# B&R Automation Studio project DietrichBrewing
Automation Studio 4.12.3.127 SP; technology packages: Acp10Arnc0 5.19.1, mapp 5.19.0, mappControl 5.19.0, mappView 5.19.0

## Configuration Config1

CPU X20CP0482, AutomationRuntime B4.93, Build 4.1.2, Safety 0.0, Vc V4.72.6

### Task classes (Cpu.sw)
```
Cyclic#1 (cycle 1000 us, tolerance 0 us):
  KettleCont <- ProcessControl.KettleControl.prg
Cyclic#2 (cycle 20000 us, tolerance 20000 us):
  HLTControl <- ProcessControl.HLTControl.prg
Cyclic#4 (cycle 100000 us, tolerance 100000 us):
  BrewingSeq <- Brewing.BrewingSeq.prg
  HMIProgram <- HMIControl.HMIProgram.prg
  MashTunCon <- ProcessControl.MashTunControl.prg
Binaries: FWRules, arsvcreg, TCData, udbdef, mvLoader, User, iomap, Config, Role, arconfig, asfw, ashwac, sysconf, ashwd, Config_1
Libraries: MpTemp, MpBase, MTBasics, brsystem, sys_lib, MTTypes, runtime, Functions, standard, asieccon, arssl, AsIODiag, Acp10man, Acp10par, NcGlobal, ViBase, AsZip, FileIO, AsARCfg, powerlnk, AsEPL, AsIO, astime, SfDomain, CoTrace
```

### Hardware
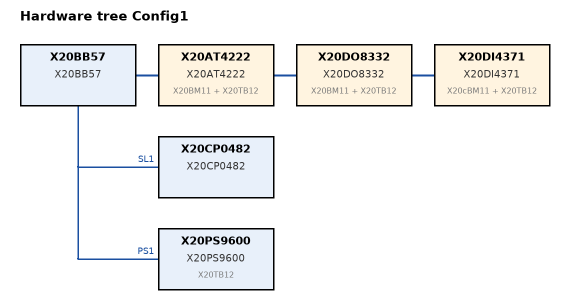
```
X20AT4222 : X20AT4222 v1.4.0.0  [SS1 -> X20TB12a.SS; SL -> X20BM11.SL1]
  InputFilter = 1ms
X20BB57 : X20BB57 v1.2.0.0
X20BM11 : X20BM11 v1.1.0.0  [X2X1 -> X20BB57.IF6]
X20BM11a : X20BM11 v1.1.0.0  [X2X1 -> X20BM11.X2X2]
X20CP0482 : X20CP0482 v1.7.0.0  [SL -> X20BB57.SL1]
  Connector IF2:
    ActivateDevice = 1
    Mode = Manual
    InternetAddress = 192.168.4.64
    SubnetMask = 255.255.255.0
  Connector IF3:
    ActivatePowerlink = 0
  ConfigurationID = DietrichBrewing_Config1
  TimerDeviceType = SWIOTIMER
  SystemTick = 1000
  Cyclic1Duration = 1000
  Cyclic1Tolerance = 0
  Cyclic2Duration = 20000
  Cyclic2Tolerance = 20000
  Cyclic3Duration = 50000
  Cyclic3Tolerance = 50000
  Cyclic4Duration = 100000
  Cyclic4Tolerance = 100000
  Cyclic5Duration = 200000
  Cyclic5Tolerance = 200000
  Cyclic6Duration = 500000
  Cyclic6Tolerance = 500000
  Cyclic7Duration = 1000000
  Cyclic7Tolerance = 1000000
  Cyclic8Duration = 10000
  Cyclic8Tolerance = 30000000
  FileDevice1
  FileDeviceName1 = USER
  FileDevicePath1 = USER_PATH
  ActivateOpcUa = 1
  OpcUaInformationModels_PV_Version = 1
X20DI4371 : X20DI4371 v1.2.0.0  [SS1 -> X20TB12c.SS; SL -> X20cBM11.SL1]
  Supervision = off
X20DO8332 : X20DO8332 v1.5.0.0  [SS1 -> X20TB12b.SS; SL -> X20BM11a.SL1]
X20PS9600 : X20PS9600 v1.6.0.0  [PS -> X20BB57.PS1; SS1 -> X20TB12.SS]
X20TB12 : X20TB12 v1.0.0.0
X20TB12a : X20TB12 v1.0.0.0
X20TB12b : X20TB12 v1.0.0.0
X20TB12c : X20TB12 v1.0.0.0
X20cBM11 : X20cBM11 v1.1.0.0  [X2X1 -> X20BM11a.X2X2]
```

### IoMap.iom - X20CP0482/IoMap.iom
```iecst
VAR_CONFIG
	::HLTHeater AT %QX."X20DO8332".DigitalOutput01;
	::KettleHeater AT %QX."X20DO8332".DigitalOutput02;
	::HLTPump AT %QX."X20DO8332".DigitalOutput03;
	::MashPump AT %QX."X20DO8332".DigitalOutput04;
	::Buzzer AT %QX."X20DO8332".DigitalOutput05;
	::ValveSelector AT %QX."X20DO8332".DigitalOutput06;
	::ValveOff AT %QX."X20DO8332".DigitalOutput07;
	::ValveOn AT %QX."X20DO8332".DigitalOutput08;
END_VAR
```

### Acp10cfg.ncc - X20CP0482/Motion/Acp10cfg.ncc
```
NcConfiguration (Version=5.16.2, NcSwId=Acp10)
  ACP10CF1_typ:
    cnt_nettrc_rec_drive = 150
    bufsize_trace_upload = 1200
    tc_nc_man_task = Cyclic #1
    glob_pv_as_ncobject = Yes
    ncsys_dl_broadcast = Yes
    ncsys_dl_acp_reset = Yes
    safemc_log_err_to_ax = Yes
    network_init:
      ncsw_init_execute = Yes
      automatic_execute = No
      node_nr_warning = Yes
      net_err_before_ncact = Yes
    nettrc:
      enter_parsecrec = Yes
      enter_ncaction = Yes
      save_ring_startidx = No
    cam_prof_download:
      cam_dat_dl_parallel = No
      tc_cam_dl_parallel = Task class for NC Manager task
```

### Config.tempcontroller - X20CP0482/mappControl/Config.tempcontroller
```
Element Cfg_HLTTemp (Type=tempcontroller)
  TempController:
    PWMParameters:
      Heat:
        Period = 0.5
  Alarms:
    UserAlarm = Yes
Element Cfg_KettleTemp (Type=tempcontroller)
  Alarms:
    UserAlarm = Yes
```

## Logical view

Binary libraries used (declarations not repeated): operator, runtime, astime, AsIecCon, brsystem, sys_lib, MTTypes, standard, AsIODiag, ViBase, AsZip, FileIO, AsARCfg, powerlnk, AsEPL, AsIO, CoTrace, Acp10man 5.19.1, Acp10par 5.19.1, NcGlobal 5.19.1, MpAlarmX, MpBase, MpTemp 5.19.0, MTBasics

### Global.typ - Global data types
```iecst
(*Main Type*)

TYPE
	MashToHLT : 	STRUCT
		Start : BOOL;
		HLTTemp : REAL;
	END_STRUCT;
	ProcControl : 	STRUCT
		setPower : REAL;
		currPower : REAL;
		currTemp : REAL;
		SetTemp : REAL;
		TempCtrl : TempCont;
		State : ControlState;
		Status : SystemStatus;
		i : SystemInput;
	END_STRUCT;
END_TYPE

(*HMI Inputs and Status*)

TYPE
	SystemInput : 	STRUCT
		ResetError : BOOL;
		EStop : BOOL;
		Auto : BOOL;
		Stop : BOOL;
		Pause : BOOL;
		Start : BOOL;
	END_STRUCT;
	SystemStatus : 	STRUCT
		Automatic : BOOL;
		Manual : BOOL;
		Running : BOOL;
		Stopped : BOOL;
		Paused : BOOL;
		On : BOOL;
	END_STRUCT;
END_TYPE

(*Temp Controller Types*)

TYPE
	TempCont : 	STRUCT
		Ctrl : MpTempController;
		Ptr : MpTempControllerParType;
		PWM : MTBasicsPWM;
	END_STRUCT;
END_TYPE

(*State Machines*)

TYPE
	ControlState :
		(
		Stop,
		Manual,
		Automatic
		);
END_TYPE
```

### Global.var - Global variables
```iecst
(*Between Programs*)
VAR
	FromMashCyc : MashToHLT;
END_VAR
(*Output Mapping*)
VAR
	Buzzer : BOOL;
	ValveSelector : BOOL; (*Off = Mash, On = HLT*)
	ValveOff : BOOL;
	ValveOn : BOOL;
	SysPower : BOOL;
	HLTPump : BOOL;
	MashPump : BOOL;
	CoolingPump : BOOL;
	HLTHeater : BOOL;
	KettleHeater : BOOL;
END_VAR
(*Temperature Controller Variables*)
VAR
	rawMashTemp : INT;
	rawKettleTemp : INT;
	rawHLTTemp : INT;
END_VAR
```

### Package Logical/Libraries - Global libraries

### Library Logical/Libraries/Functions (IEC)

#### Functions.fun - Exported functions and function blocks
```iecst
{REDUND_ERROR} FUNCTION Device : BOOL (*TODO: Add your comment here*) (*$GROUP=User,$CAT=User,$GROUPICON=User.png,$CATICON=User.png*)
	VAR_INPUT
		AutoMode : BOOL;
		AutoExpected : BOOL;
		pbExpected : BOOL;
	END_VAR
	VAR_IN_OUT
		Output : BOOL;
	END_VAR
	VAR
		Expected : BOOL;
	END_VAR
END_FUNCTION
```

#### Device.st
```iecst
//Set device on or off with HMI or sequence
FUNCTION Device

	IF NOT AutoMode THEN

		//Manual Operation
		IF pbExpected  THEN
			Expected  := TRUE;
		ELSIF NOT pbExpected THEN
			Expected  := FALSE;
		END_IF

	ELSE
		//Auto operation
		IF AutoExpected THEN
			Expected:= TRUE;
		ELSIF NOT AutoExpected THEN
			Expected := FALSE;
		END_IF
	END_IF

	//Set output of function
	Output := Expected;
END_FUNCTION
```

### Program Logical/Brewing/BrewingSeq (IEC)

#### Types.typ
```iecst
TYPE
	Seq :
		(
		Reset,
		FillTanks,
		PreHeat,
		Mash,
		Boil
		);
END_TYPE
```

#### Variables.var
```iecst
VAR
	HeatTime : TON;
	Sequence : Seq;
	pbMashPump : BOOL;
END_VAR
```

#### Main.st
```iecst
PROGRAM _INIT

END_PROGRAM

PROGRAM _CYCLIC

END_PROGRAM

PROGRAM _EXIT
	(* Insert code here *)

END_PROGRAM
```

### Program Logical/Brewing/HLTControl

#### Variables.var
```iecst
VAR
	PumpExp : BOOL;
	Proc : ProcControl;
END_VAR
```

#### Main.st
```iecst
PROGRAM _INIT

END_PROGRAM

PROGRAM _CYCLIC
	//Initilize Temp Controller FB
	Proc.TempCtrl.Ctrl.Parameters := ADR(Proc.TempCtrl.Ptr);
	Proc.TempCtrl.Ctrl.MpLink := ADR(Cfg_HLTTemp);

	//Mash cycle variables
	IF EDGEPOS(FromMashCyc.Start) THEN
		Proc.i.Auto 	:= TRUE;
		Proc.i.Start 	:= TRUE;
		Proc.SetTemp 	:= FromMashCyc.HLTTemp;
	ELSIF EDGENEG(FromMashCyc.Start) THEN
		Proc.i.Auto 	:= FALSE;
		Proc.i.Start 	:= FALSE;
	END_IF

	//Automatic and manual conditions
	Proc.Status.Automatic 	:= Proc.i.Auto;
	Proc.Status.Manual		:= NOT Proc.i.Auto;

	//Map Variables
	Proc.TempCtrl.Ctrl.Control := Proc.i.Start;
	Proc.TempCtrl.Ctrl.ErrorReset := Proc.i.ResetError;
	Proc.TempCtrl.Ctrl.SetTemperature := Proc.SetTemp;

	IF Proc.Status.Automatic THEN
		Proc.State := Automatic;
	ELSIF Proc.Status.Manual THEN
		Proc.State := Manual;
	END_IF

	//Set the state machine
	IF  DiagCpuIsARsim() OR DiagCpuIsSimulated() THEN
		Proc.currTemp := Proc.TempCtrl.Ctrl.Info.Simulation.ActualTemperature;
		Proc.currPower := Proc.TempCtrl.Ctrl.Info.Simulation.HeatValue;
		Proc.TempCtrl.Ctrl.Simulate := TRUE;
	ELSE
		Proc.TempCtrl.Ctrl.ActualTemperature := rawHLTTemp * 1000;

		Proc.currTemp	:= rawHLTTemp * 1000;
		Proc.TempCtrl.Ctrl.Simulate := FALSE;
	END_IF

	//Temperature controller state machine
	CASE Proc.State OF

		Automatic:
			//Temperature control parameters
			Proc.TempCtrl.PWM.Enable 	:= FALSE;
			Proc.TempCtrl.Ctrl.Enable 	:= TRUE;

			//HMI Variables
			HLTHeater := Proc.TempCtrl.Ctrl.Heat;
			Proc.currPower 	:= Proc.TempCtrl.Ctrl.HeatValue;

		Manual:
			//Temperature control parmeters
			Proc.TempCtrl.PWM.Enable 	:= Proc.i.Start;
			Proc.TempCtrl.Ctrl.Enable 	:= FALSE;
			Proc.TempCtrl.PWM.DutyCycle := Proc.setPower;
			Proc.TempCtrl.PWM.MinPulseWidth := 0.1;
			Proc.TempCtrl.PWM.Period := 1.0;

			//HMI Variables
			HLTHeater := Proc.TempCtrl.PWM.Out;
			IF Proc.TempCtrl.PWM.Active THEN
				Proc.currPower := Proc.TempCtrl.PWM.DutyCycle;
			ELSE
				Proc.currPower := 0;
			END_IF

	END_CASE

	//Call FB's
	Proc.TempCtrl.Ctrl();
	Proc.TempCtrl.PWM();

	//Set pump output
	HLTPump := PumpExp;
END_PROGRAM

PROGRAM _EXIT
	(* Insert code here *)

END_PROGRAM
```

### Program Logical/Brewing/KettleControl (IEC)

#### Main.st - Init, cyclic, exit code
```iecst
PROGRAM _INIT
	(* Insert code here *)

END_PROGRAM

PROGRAM _CYCLIC
	//Initilize Temp Controller FB
	Proc.TempCtrl.Ctrl.Parameters := ADR(Proc.TempCtrl.Ptr);
	Proc.TempCtrl.Ctrl.MpLink := ADR(Cfg_KettleTemp);
	//Map Variables
	Proc.TempCtrl.Ctrl.Control := Proc.i.Start;
	Proc.TempCtrl.Ctrl.ErrorReset := Proc.i.ResetError;

	//Automatic and manual conditions
	Proc.Status.Automatic 	:= Proc.i.Auto;
	Proc.Status.Manual		:= NOT Proc.i.Auto;

	IF Proc.Status.Automatic THEN
		Proc.State := Automatic;
	ELSIF Proc.Status.Manual THEN
		Proc.State := Manual;
	ELSE
	;
	END_IF

	//Set the state machine
	IF  DiagCpuIsARsim() OR DiagCpuIsSimulated() THEN
		Proc.TempCtrl.Ctrl.Enable	:= TRUE;
		Proc.TempCtrl.Ctrl.Simulate := TRUE;
		Proc.currTemp := Proc.TempCtrl.Ctrl.Info.Simulation.ActualTemperature;
	ELSE
		Proc.currTemp := rawHLTTemp * 1000;
	END_IF

	//Temperature controller state machine
	CASE Proc.State OF

		Manual:
			//PWM control
			Proc.TempCtrl.PWM.Enable 	:= Proc.i.Start;

			//PWM Parameters
			Proc.TempCtrl.PWM.DutyCycle := Proc.setPower;
			Proc.TempCtrl.PWM.MinPulseWidth := 0.1;
			Proc.TempCtrl.PWM.Period 		:= 1.0;
			KettleHeater := Proc.TempCtrl.PWM.Out;

			//HMI Variables
			IF Proc.TempCtrl.PWM.Active THEN
				Proc.currPower := Proc.TempCtrl.PWM.DutyCycle;
			ELSE
				Proc.currPower := 0;
			END_IF

		Automatic:
			//Not Used

	END_CASE

	//Call Action Files
	Displayclock;
	PowerControl;

	//Call FB's
	Proc.TempCtrl.Ctrl();
	Proc.TempCtrl.PWM();
	KettleTmr();
END_PROGRAM

PROGRAM _EXIT
	(* Insert code here *)

END_PROGRAM
```

#### Variables.var - Local variables
```iecst
(*Hop Control Variables*)
VAR
	SelectedHopTime : USINT;
	HopTime : ARRAY[0..5] OF USINT;
	i : INT;
	currHop : INT;
	remainTime : USINT;
END_VAR
(*Kettle Control*)
VAR
	Proc : ProcControl;
	KettleTmr : TON;
	TimePre : TIME;
	StartKettle : BOOL;
	TmrDT : TIMEStructure;
	HrRe : STRING[4];
	MinRe : STRING[4];
	SecRe : STRING[4];
	TmrRemain : STRING[10];
	pbFastDown : BOOL;
	pbFastUp : BOOL;
	pbUp : BOOL;
	pbDown : BOOL;
	HopSelection : DINT;
	PrevSelection : DINT;
	PrevHopTime : DINT;
END_VAR
```

#### Displayclock.st
```iecst
ACTION Displayclock:

	//Kettle timer
	KettleTmr.PT := DINT_TO_TIME(TimePre*60000);
	//Start Kettle Timer
	KettleTmr.IN := StartKettle;

	//Calculate and display the remaining time
	TIME_TO_TIMEStructure((KettleTmr.PT - KettleTmr.ET), ADR(TmrDT));
	HrRe 	:= USINT_TO_STRING(TmrDT.hour);
	MinRe 	:= USINT_TO_STRING(TmrDT.minute);
	SecRe	:= USINT_TO_STRING(TmrDT.second);
	TmrRemain := CONCAT(HrRe, ':');
	TmrRemain := CONCAT(TmrRemain, MinRe);
	TmrRemain := CONCAT(TmrRemain,':');
	TmrRemain := CONCAT(TmrRemain, SecRe);

	//Kettle Time is Done Rest Everything
	IF KettleTmr.Q THEN
		StartKettle := FALSE;
		Proc.i.Start := FALSE;
		Buzzer := TRUE;
	END_IF

END_ACTION
```

#### HopControl.st
```iecst
ACTION HopControl:

	//Detect Changed value
	IF SelectedHopTime <> PrevHopTime THEN
		HopTime[HopSelection] := SelectedHopTime;
		PrevHopTime := SelectedHopTime;
	END_IF

	//Detect new selection
	IF HopSelection <> PrevSelection THEN
		SelectedHopTime := HopTime[HopSelection];
		PrevSelection := HopSelection;
	END_IF

	FOR i := 1 TO 5 DO
		IF KettleTmr.IN THEN
			//Determine current addition
			IF TmrDT.minute < HopTime[i] AND TmrDT.second = 0 THEN
				currHop := i;
				Buzzer := TRUE;
			END_IF

			//Determine time for next addition
			remainTime := TmrDT.minute - HopTime[currHop + 1] +1;
		ELSE
			currHop := 0;
		END_IF
	END_FOR;

END_ACTION
```

#### PowerControl.st - not listed in the package file held
```iecst
ACTION PowerControl:

	IF Proc.TempCtrl.PWM.Active THEN

		IF pbUp THEN
			Proc.setPower := Proc.setPower + 5;
			pbUp := FALSE;
		END_IF

		IF pbDown THEN
			Proc.setPower := Proc.setPower - 5;
			pbDown := FALSE;
		END_IF
	END_IF

END_ACTION
```

### Program Logical/Brewing/MashTunControl

#### Main.st
```iecst
PROGRAM _INIT
		//Initilize Temp Controller FB
	mProc.TempCtrl.Ctrl.Parameters := ADR(mProc.TempCtrl.Ptr);
	mProc.TempCtrl.Ctrl.MpLink := ADR(Cfg_MashTemp_simulated);

END_PROGRAM

PROGRAM _CYCLIC

		//Automatic and manual conditions
	mProc.Status.Automatic 	:= mProc.i.Start;
	mProc.Status.Manual		:= NOT mProc.i.Start;
	FromMashCyc.Start := mProc.i.Start;

	IF mProc.Status.Automatic THEN
		mProc.State := Automatic;
	ELSIF mProc.Status.Manual THEN
		mProc.State := Manual;
	END_IF

	//Simulate Values
	IF  DiagCpuIsARsim() OR DiagCpuIsSimulated() THEN
		mProc.currTemp := mProc.TempCtrl.Ctrl.Info.Simulation.ActualTemperature;
		mProc.TempCtrl.Ctrl.Simulate := TRUE;
		mProc.TempCtrl.PWM.Enable := FALSE;
		mProc.TempCtrl.Ctrl.Enable := TRUE;
		mProc.TempCtrl.Ctrl.SetTemperature := mProc.SetTemp;
		mProc.TempCtrl.Ctrl.Control := mProc.i.Start;
	ELSE
		mProc.currTemp := rawMashTemp / 1000;
		mProc.TempCtrl.Ctrl.Simulate := FALSE;
	END_IF

	//Turn off pump when switching auto and manual
	IF EDGENEG(mProc.i.Start) THEN
		pbMashPump 		:= FALSE;
		StartMash 		:= FALSE;
		MashTmr.IN		:= FALSE;
		mProc.i.Start 	:= FALSE;
	END_IF

	CASE mProc.State OF

		Manual:
			//Figure out how to simulate the temperature
			mProc.currTemp := rawMashTemp / 1000;
			PumpExp := pbMashPump;

		Automatic:

			//Set parameters
			FromMashCyc.HLTTemp := mProc.SetTemp + 3;
			pbMashPump := PumpExp;

			//Stop pump if the mash temp gets too high
			IF mProc.currTemp > (mProc.SetTemp * 1.10) THEN
				PumpExp	:= FALSE;
			ELSE
				PumpExp	:= TRUE;
			END_IF

	END_CASE

	//Mash timer
	MashTmr.PT := DINT_TO_TIME(TimePre*60000);
	MashTmr.IN := StartMash;

	//Mash Time is Done Rest Everything
	IF MashTmr.Q THEN
		StartMash := FALSE;
		mProc.i.Start := FALSE;
		Buzzer := TRUE;
	END_IF

	//Calculate and display the remaining time
	TIME_TO_TIMEStructure((MashTmr.PT - MashTmr.ET), ADR(TmrDT));
	HrRe 	:= USINT_TO_STRING(TmrDT.hour);
	MinRe 	:= USINT_TO_STRING(TmrDT.minute);
	SecRe	:= USINT_TO_STRING(TmrDT.second);
	TmrRemain := CONCAT(HrRe, ':');
	TmrRemain := CONCAT(TmrRemain, MinRe);
	TmrRemain := CONCAT(TmrRemain,':');
	TmrRemain := CONCAT(TmrRemain, SecRe);

	//HMI Control
	MashPump := PumpExp;

	//Call Function Blocks
	MashTmr();

	//call simulated FUB
	mProc.TempCtrl.Ctrl();
	mProc.TempCtrl.PWM();

END_PROGRAM

PROGRAM _EXIT
	(* Insert code here *)

END_PROGRAM
```

### Program Logical/FillingTanks/FillingTanks (IEC)

#### Main.st - Init, cyclic, exit code
```iecst
PROGRAM _INIT
	ValveTmr.PT := T#2s;
END_PROGRAM

PROGRAM _CYCLIC

	//Start and stop logic
	IF  DiagCpuIsARsim() OR DiagCpuIsSimulated() THEN
		SimFlowMeter;
	END_IF

	//Fill tank programs
	FillHLT;
	FillMash;

	//Control Selector Relay
	IF AutoFillHLT.Valve THEN
		ValveSelector := TRUE;
	END_IF

	//Open or close valve
	IF EDGEPOS(AutoFillHLT.Valve OR AutoFillMash.Valve) THEN
		ValveOn := TRUE;
		ValveTmr.IN := TRUE;
	ELSIF EDGENEG(AutoFillHLT.Valve OR AutoFillMash.Valve) THEN
		ValveOff := TRUE;
		ValveTmr.IN := TRUE;
	END_IF

	IF ValveTmr.Q THEN
		ValveOn := FALSE;
		ValveOff := FALSE;
		ValveTmr.IN := FALSE;
		ValveSelector := FALSE;
	END_IF

	ValveTmr();
END_PROGRAM

PROGRAM _EXIT

END_PROGRAM
```

#### Types.typ - Local data types
```iecst
TYPE
	ValveControl : 	STRUCT
		Reset : BOOL;
		Stop : BOOL;
		Start : BOOL;
		ValveR : R_TRIG;
		Valve : BOOL;
		VolumePV : REAL;
		VolumeSP : REAL;
		State : ControlState;
	END_STRUCT;
END_TYPE
```

#### Variables.var - Local variables
```iecst
VAR
	HLTFillLevel : REAL;
	MashFillLevel : REAL;
	ValveTmr : TON;
	AutoFillMash : ValveControl;
	AutoFillHLT : ValveControl;
	MashImgCont : INT;
	HLTImgCont : INT;
END_VAR
(*Simulation Variables*)
VAR
	SimFlowMeterPulse : TON;
	SimFlowMeterVal : REAL;
END_VAR
```

#### SimFlowMeter.st
```iecst
ACTION SimFlowMeter:

	SimFlowMeterPulse.PT := T#100ms;
	IF (AutoFillHLT.Valve) THEN
		SimFlowMeterPulse.IN	:= TRUE;
		IF(SimFlowMeterPulse.Q) THEN
			SimFlowMeterPulse.IN := FALSE;
			//Simulated accumulated value
			SimFlowMeterVal := SimFlowMeterVal + 0.1;
		END_IF
	END_IF

	SimFlowMeterPulse();

END_ACTION
```

#### FillHLT.st
```iecst
ACTION FillHLT:
	//Start and stop logic
	IF AutoFillHLT.Start THEN
		AutoFillHLT.State := Automatic;
	ELSIF AutoFillHLT.Stop THEN
		AutoFillHLT.State := Stop;
	END_IF

	//Image animation
	IF AutoFillHLT.VolumePV > AutoFillHLT.VolumeSP / 4 AND (AutoFillHLT.VolumePV < AutoFillHLT.VolumeSP / 2) THEN
		HLTImgCont := 1;
	ELSIF AutoFillHLT.VolumePV >= AutoFillHLT.VolumeSP / 2 AND (AutoFillHLT.VolumePV < AutoFillHLT.VolumeSP ) THEN
		HLTImgCont := 2;
	ELSIF AutoFillHLT.VolumePV >= AutoFillHLT.VolumeSP THEN
		HLTImgCont := 3;
	ELSE
		HLTImgCont := 0;
	END_IF

	CASE AutoFillHLT.State OF

		Stop:
			AutoFillHLT.Valve	:= FALSE;
			AutoFillHLT.Stop	:= FALSE;
			AutoFillHLT.State 	:= Manual;

		Automatic:

			IF AutoFillHLT.Start AND (AutoFillHLT.VolumePV < AutoFillHLT.VolumeSP) THEN
				AutoFillHLT.Valve 	:= TRUE;
			ELSE
				AutoFillHLT.Start := FALSE;
				AutoFillHLT.State := Stop;
			END_IF

		Manual:
			//Manual Control of Valve
			IF AutoFillHLT.Reset THEN
				AutoFillHLT.Reset	:= FALSE;
				AutoFillHLT.VolumePV := 0.0;
			END_IF

	END_CASE

END_ACTION
```

#### FillMash.st
```iecst
ACTION FillMash:

	//Start and stop logic
	IF(AutoFillMash.Start) THEN
		AutoFillMash.State := Automatic;
	ELSIF AutoFillMash.Stop THEN
		AutoFillMash.State := Stop;
	END_IF

	//Image animation
	IF AutoFillMash.VolumePV > AutoFillMash.VolumeSP / 4 AND (AutoFillMash.VolumePV < AutoFillMash.VolumeSP / 2) THEN
		MashImgCont := 1;
	ELSIF AutoFillMash.VolumePV >= AutoFillMash.VolumeSP / 2 AND (AutoFillMash.VolumePV < AutoFillMash.VolumeSP ) THEN
		MashImgCont := 2;
	ELSIF AutoFillMash.VolumePV >= AutoFillMash.VolumeSP THEN
		MashImgCont := 3;
	ELSE
		MashImgCont := 0;
	END_IF

	CASE AutoFillMash.State OF

		Stop:
			AutoFillMash.Valve	:= FALSE;
			AutoFillMash.Stop	:= FALSE;
			AutoFillMash.State 	:= Manual;

		Automatic:

			IF AutoFillMash.Start AND (AutoFillMash.VolumePV < AutoFillMash.VolumeSP) THEN
				AutoFillMash.Valve 	:= TRUE;
			ELSE
				AutoFillMash.Start := FALSE;
				AutoFillMash.State := Stop;
			END_IF

		Manual:

			IF AutoFillMash.Reset THEN
				AutoFillMash.VolumePV := 0.0;
				AutoFillMash.Reset	:= FALSE;
			END_IF

	END_CASE

END_ACTION
```

### Program Logical/HMIControl/HMIProgram (IEC)

#### Variables.var
```iecst
VAR
	TestBuzzer : BOOL;
	FlashOn : TON;
	FlashOff : TON;
	SlienceVis : BOOL;
	SlienceBtn : BOOL;
END_VAR
```

#### Main.st
```iecst
PROGRAM _INIT
	(* Insert code here *)
	FlashOn.PT := T#1000ms;
	FlashOff.PT := T#500ms;
END_PROGRAM

PROGRAM _CYCLIC

	//Code Stored Here to Drive HMI Functions

	//Buzzer Slience Logic
	IF Buzzer THEN
		SlienceVis := FlashOn.IN;
	END_IF

	IF FlashOn.Q THEN
		FlashOn.IN := FALSE;
		FlashOff.IN := TRUE;
	ELSIF FlashOff.Q OR EDGEPOS(Buzzer) THEN
		FlashOn.IN := TRUE;
		FlashOff.IN := FALSE;
	END_IF

	IF SlienceBtn THEN
		Buzzer := FALSE;
		FlashOff.IN := FALSE;
		FlashOn.IN := FALSE;
		SlienceVis := FALSE;
		SlienceBtn := FALSE;
	END_IF

	//Call Function Blocks
	FlashOn();
	FlashOff();

END_PROGRAM

PROGRAM _EXIT
	(* Insert code here *)

END_PROGRAM
```

- Visualisation Logical/mappView (not shown)

### Program Logical/Fermenting/Fermenting (IEC)

#### ChillerControl.st
```iecst
ACTION ChillerControl:

END_ACTION
```

### Program Logical/ProcessControl/HLTControl (IEC)

#### Variables.var
```iecst
VAR
	Proc : ProcControl;
END_VAR
```

#### Main.st
```iecst
PROGRAM _INIT

END_PROGRAM

PROGRAM _CYCLIC
	//Initilize Temp Controller FB
	Proc.TempCtrl.Ctrl.Parameters := ADR(Proc.TempCtrl.Ptr);
	Proc.TempCtrl.Ctrl.MpLink := ADR(Cfg_HLTTemp);
	//Map Variables
	Proc.TempCtrl.Ctrl.Control := Proc.i.Start;
	Proc.TempCtrl.Ctrl.ErrorReset := Proc.i.ResetError;

	//Mash cycle variables
	IF EDGEPOS(FromMashCyc.Start) THEN
		Proc.i.Auto 	:= TRUE;
		Proc.i.Start 	:= TRUE;
		Proc.SetTemp 	:= FromMashCyc.HLTTemp;
	ELSIF EDGENEG(FromMashCyc.Start) THEN
		Proc.i.Auto 	:= FALSE;
		Proc.i.Start 	:= FALSE;
	END_IF

	//Automatic and manual conditions
	Proc.Status.Automatic 	:= Proc.i.Auto;
	Proc.Status.Manual		:= NOT Proc.i.Auto;

	//Set the state machine
	IF  DiagCpuIsARsim() OR DiagCpuIsSimulated() THEN
		IF Proc.Status.Automatic THEN
			Proc.State := SimAuto;
		ELSIF Proc.Status.Manual THEN
			Proc.State := SimManual;
		END_IF
	END_IF

	//Temperature controller state machine
	CASE Proc.State OF

		SimAuto:
			//Setup variables
			Proc.TempCtrl.PWM.Enable := FALSE;
			Proc.TempCtrl.Ctrl.Enable := TRUE;
			Proc.TempCtrl.Ctrl.Simulate := TRUE;
			//Map Simulated Values
			Proc.TempCtrl.Ctrl.ActualTemperature := Proc.TempCtrl.Ctrl.Info.Simulation.ActualTemperature;
			Proc.TempCtrl.Ctrl.SetTemperature := Proc.SetTemp;
			Proc.TempCtrl.Ctrl.Control := Proc.i.Start;
			Proc.currTemp := Proc.TempCtrl.Ctrl.Info.Simulation.ActualTemperature;
			Proc.currPower := Proc.TempCtrl.Ctrl.Info.Simulation.HeatValue;
			HLTHeater := Proc.TempCtrl.Ctrl.Info.Simulation.Heat;

		SimManual:
			Proc.TempCtrl.PWM.Enable 	:= TRUE;
			Proc.TempCtrl.Ctrl.Enable	:= FALSE;
			//Proc.TempCtrl.PWM Variables
			Proc.TempCtrl.PWM.DutyCycle := Proc.setPower;
			Proc.TempCtrl.PWM.MinPulseWidth := 0.1;
			Proc.TempCtrl.PWM.Period 		:= 1.0;

		Automatic:
			Proc.TempCtrl.PWM.Enable 	:= TRUE;
			Proc.TempCtrl.Ctrl.Enable 	:= FALSE;
			Proc.TempCtrl.Ctrl.ActualTemperature := rawHLTTemp * 1000;
			Proc.currPower 	:= Proc.TempCtrl.Ctrl.HeatValue;
			Proc.currTemp	:= rawHLTTemp * 1000;

		Manual:
			Proc.TempCtrl.PWM.Enable 	:= FALSE;
			Proc.TempCtrl.Ctrl.Enable 	:= TRUE;
			//Proc.TempCtrl.PWM Variables
			Proc.TempCtrl.PWM.DutyCycle := Proc.setPower;
			Proc.TempCtrl.PWM.MinPulseWidth := 0.1;
			Proc.TempCtrl.PWM.Period := 1.0;
			Proc.currTemp := rawHLTTemp * 1000;

	END_CASE

	//Call FB's
	Proc.TempCtrl.Ctrl();
	Proc.TempCtrl.PWM();
END_PROGRAM

PROGRAM _EXIT
	(* Insert code here *)

END_PROGRAM
```

### Program Logical/ProcessControl/MashTunControl (IEC)

#### Main.st
```iecst
PROGRAM _INIT
	(* Insert code here *)

END_PROGRAM

PROGRAM _CYCLIC

		//Automatic and manual conditions
	mProc.Status.Automatic 	:= mProc.i.Start;
	mProc.Status.Manual		:= NOT mProc.i.Start;
	FromMashCyc.Start := mProc.i.Start;

	//Set the state machine
	IF  DiagCpuIsARsim() OR DiagCpuIsSimulated() THEN
		IF mProc.Status.Automatic THEN
			mProc.State := SimAuto;
		ELSIF mProc.Status.Manual THEN
			mProc.State := SimManual;
		END_IF
	END_IF

	//Turn off pump when switching auto and manual
	IF EDGENEG(mProc.i.Start) THEN
		pbMashPump 		:= FALSE;
		StartMash 		:= FALSE;
		MashTmr.IN		:= FALSE;
		mProc.i.Start 	:= FALSE;
	END_IF

	CASE mProc.State OF

		SimManual:
			//Figure out how to simulate the temperature
			mProc.currTemp := rawMashTemp / 1000;
			PumpExp := pbMashPump;

		SimAuto:
			//Figure out how to simulate the temperature
			mProc.currTemp := rawMashTemp / 1000;
			FromMashCyc.HLTTemp := mProc.SetTemp + 15;
			pbMashPump := PumpExp;

			//Stop pump if the mash temp gets too high
			IF mProc.currTemp < mProc.SetTemp THEN
				PumpExp	:= TRUE;
			ELSE
				PumpExp	:= FALSE;
			END_IF

			//Mash timer
			MashTmr.PT := DINT_TO_TIME(TimePre*60000);
			//Start Mash Timer
			MashTmr.IN := StartMash;

			//Calculate and display the remaining time
			TIME_TO_TIMEStructure((MashTmr.PT - MashTmr.ET), ADR(TmrDT));
			HrRe 	:= USINT_TO_STRING(TmrDT.hour);
			MinRe 	:= USINT_TO_STRING(TmrDT.minute);
			SecRe	:= USINT_TO_STRING(TmrDT.second);
			TmrRemain := CONCAT(HrRe, ':');
			TmrRemain := CONCAT(TmrRemain, MinRe);
			TmrRemain := CONCAT(TmrRemain,':');
			TmrRemain := CONCAT(TmrRemain, SecRe);

			//Mash Time is Done Rest Everything
			IF MashTmr.Q THEN
				StartMash := FALSE;
				mProc.i.Start := FALSE;
			END_IF

		Manual:

			mProc.currTemp := rawMashTemp / 1000;

	END_CASE

	MashPump := PumpExp;

	MashTmr();
END_PROGRAM

PROGRAM _EXIT
	(* Insert code here *)

END_PROGRAM
```

### Program Logical/ProcessControl/KettleControl (IEC)

#### Main.st
```iecst
PROGRAM _INIT
	(* Insert code here *)

END_PROGRAM

PROGRAM _CYCLIC
	//Initilize Temp Controller FB
	Proc.TempCtrl.Ctrl.Parameters := ADR(Proc.TempCtrl.Ptr);
	Proc.TempCtrl.Ctrl.MpLink := ADR(Cfg_KettleTemp);
	//Map Variables
	Proc.TempCtrl.Ctrl.Control := Proc.i.Start;
	Proc.TempCtrl.Ctrl.ErrorReset := Proc.i.ResetError;

	//Automatic and manual conditions
	Proc.Status.Automatic 	:= Proc.i.Auto;
	Proc.Status.Manual		:= NOT Proc.i.Auto;

	//Set the state machine
	IF  DiagCpuIsARsim() OR DiagCpuIsSimulated() THEN
		IF Proc.Status.Automatic THEN
			Proc.State := SimAuto;
		ELSIF Proc.Status.Manual THEN
			Proc.State := SimManual;
		END_IF
	END_IF

	//Temperature controller state machine
	CASE Proc.State OF

		SimAuto:
			//Setup variables
			Proc.TempCtrl.PWM.Enable := FALSE;
			Proc.TempCtrl.Ctrl.Enable := TRUE;
			Proc.TempCtrl.Ctrl.Simulate := TRUE;
			//Map Simulated Values
			Proc.TempCtrl.Ctrl.ActualTemperature := Proc.TempCtrl.Ctrl.Info.Simulation.ActualTemperature;
			Proc.TempCtrl.Ctrl.SetTemperature := Proc.SetTemp;
			Proc.TempCtrl.Ctrl.Control := Proc.i.Start;
			Proc.currTemp := Proc.TempCtrl.Ctrl.Info.Simulation.ActualTemperature;
			Proc.currPower := Proc.TempCtrl.Ctrl.Info.Simulation.HeatValue;
			HLTHeater := Proc.TempCtrl.Ctrl.Info.Simulation.Heat;

		SimManual:
			Proc.TempCtrl.PWM.Enable 	:= TRUE;
			Proc.TempCtrl.Ctrl.Enable	:= FALSE;
			//Proc.TempCtrl.PWM Variables
			Proc.TempCtrl.PWM.DutyCycle := Proc.setPower;
			Proc.TempCtrl.PWM.MinPulseWidth := 0.1;
			Proc.TempCtrl.PWM.Period 		:= 1.0;
			Proc.currPower := Proc.TempCtrl.PWM.DutyCycle;

		Automatic:
			Proc.TempCtrl.PWM.Enable 	:= TRUE;
			Proc.TempCtrl.Ctrl.Enable 	:= FALSE;
			Proc.TempCtrl.Ctrl.ActualTemperature := rawHLTTemp * 1000;
			Proc.currPower 	:= Proc.TempCtrl.Ctrl.HeatValue;
			Proc.currTemp	:= rawHLTTemp * 1000;

		Manual:
			Proc.TempCtrl.PWM.Enable 	:= FALSE;
			Proc.TempCtrl.Ctrl.Enable 	:= TRUE;
			//Proc.TempCtrl.PWM Variables
			Proc.TempCtrl.PWM.DutyCycle := Proc.setPower;
			Proc.TempCtrl.PWM.MinPulseWidth := 0.1;
			Proc.TempCtrl.PWM.Period := 1.0;
			Proc.currTemp := rawHLTTemp * 1000;

	END_CASE

	//Kettle timer
	KettleTmr.PT := DINT_TO_TIME(TimePre*60000);
	//Start Kettle Timer
	KettleTmr.IN := StartKettle;

	//Calculate and display the remaining time
	TIME_TO_TIMEStructure((KettleTmr.PT - KettleTmr.ET), ADR(TmrDT));
	HrRe 	:= USINT_TO_STRING(TmrDT.hour);
	MinRe 	:= USINT_TO_STRING(TmrDT.minute);
	SecRe	:= USINT_TO_STRING(TmrDT.second);
	TmrRemain := CONCAT(HrRe, ':');
	TmrRemain := CONCAT(TmrRemain, MinRe);
	TmrRemain := CONCAT(TmrRemain,':');
	TmrRemain := CONCAT(TmrRemain, SecRe);

	//Kettle Time is Done Rest Everything
	IF KettleTmr.Q THEN
		StartKettle := FALSE;
		Proc.i.Start := FALSE;
	END_IF

	 	//Call FB's
	Proc.TempCtrl.Ctrl();
	Proc.TempCtrl.PWM();
	KettleTmr();
END_PROGRAM

PROGRAM _EXIT
	(* Insert code here *)

END_PROGRAM
```

### Program Logical/ProcessControl/HLT

#### Main.st
```iecst
PROGRAM _INIT

END_PROGRAM

PROGRAM _CYCLIC
	//Initilize Temp Controller FB
	Proc.TempCtrl.Ctrl.Parameters := ADR(Proc.TempCtrl.Ptr);
	Proc.TempCtrl.Ctrl.MpLink := ADR(Cfg_HLTTemp);
	//Map Variables ASasds dadasdadadawaswdawdawdsawdsawdaw
	Proc.TempCtrl.Ctrl.Control := Proc.i.Start;
	Proc.TempCtrl.Ctrl.ErrorReset := Proc.i.ResetError;

	//Mash cycle variables
	IF EDGEPOS(FromMashCyc.Start) THEN
		Proc.i.Auto 	:= TRUE;
		Proc.i.Start 	:= TRUE;
		Proc.SetTemp 	:= FromMashCyc.HLTTemp;
	ELSIF EDGENEG(FromMashCyc.Start) THEN
		Proc.i.Auto 	:= FALSE;
		Proc.i.Start 	:= FALSE;
	END_IF

	//Automatic and manual conditions
	Proc.Status.Automatic 	:= Proc.i.Auto;
	Proc.Status.Manual		:= NOT Proc.i.Auto;

	//Set the state machine
	IF  DiagCpuIsARsim() OR DiagCpuIsSimulated() THEN
		IF Proc.Status.Automatic THEN
			Proc.State := SimAuto;
		ELSIF Proc.Status.Manual THEN
			Proc.State := SimManual;
		END_IF
	END_IF

	//Temperature controller state machine
	CASE Proc.State OF

		SimAuto:
			//Setup variables
			Proc.TempCtrl.PWM.Enable := FALSE;
			Proc.TempCtrl.Ctrl.Enable := TRUE;
			Proc.TempCtrl.Ctrl.Simulate := TRUE;
			//Map Simulated Values
			Proc.TempCtrl.Ctrl.ActualTemperature := Proc.TempCtrl.Ctrl.Info.Simulation.ActualTemperature;
			Proc.TempCtrl.Ctrl.SetTemperature := Proc.SetTemp;
			Proc.TempCtrl.Ctrl.Control := Proc.i.Start;
			Proc.currTemp := Proc.TempCtrl.Ctrl.Info.Simulation.ActualTemperature;
			Proc.currPower := Proc.TempCtrl.Ctrl.Info.Simulation.HeatValue;
			HLTHeater := Proc.TempCtrl.Ctrl.Info.Simulation.Heat;

		SimManual:
			Proc.TempCtrl.PWM.Enable 	:= TRUE;
			Proc.TempCtrl.Ctrl.Enable	:= FALSE;
			//Proc.TempCtrl.PWM Variables
			Proc.TempCtrl.PWM.DutyCycle := Proc.setPower;
			Proc.TempCtrl.PWM.MinPulseWidth := 0.1;
			Proc.TempCtrl.PWM.Period 		:= 1.0;

		Automatic:
			Proc.TempCtrl.PWM.Enable 	:= TRUE;
			Proc.TempCtrl.Ctrl.Enable 	:= FALSE;
			Proc.TempCtrl.Ctrl.ActualTemperature := rawHLTTemp * 1000;
			Proc.currPower 	:= Proc.TempCtrl.Ctrl.HeatValue;
			Proc.currTemp	:= rawHLTTemp * 1000;

		Manual:
			Proc.TempCtrl.PWM.Enable 	:= FALSE;
			Proc.TempCtrl.Ctrl.Enable 	:= TRUE;
			//Proc.TempCtrl.PWM Variables
			Proc.TempCtrl.PWM.DutyCycle := Proc.setPower;
			Proc.TempCtrl.PWM.MinPulseWidth := 0.1;
			Proc.TempCtrl.PWM.Period := 1.0;
			Proc.currTemp := rawHLTTemp * 1000;

	END_CASE

	//Call FB's
	Proc.TempCtrl.Ctrl();
	Proc.TempCtrl.PWM();
END_PROGRAM

PROGRAM _EXIT
	(* Insert code here *)

END_PROGRAM
```

### Program Logical/ProcessControl/Kettle

#### Variables.var
```iecst
VAR
	Proc : ProcControl;
	KettleTmr : TON;
	TimePre : TIME;
	StartKettle : BOOL;
	TmrDT : TIMEStructure;
	HrRe : STRING[4];
	MinRe : STRING[4];
	SecRe : STRING[4];
	TmrRemain : STRING[10];
END_VAR
```

#### Main.st
```iecst
PROGRAM _INIT
	(* Insert code here *)

END_PROGRAM

PROGRAM _CYCLIC
	(* Insert code here *)
	 	//Call FB's
	Proc.TempCtrl.Ctrl();
	Proc.TempCtrl.PWM();
END_PROGRAM

PROGRAM _EXIT
	(* Insert code here *)

END_PROGRAM
```

### Program Logical/ProcessControl/MashTun

#### Variables.var
```iecst
VAR
	MashTmr : TON;
	mProc : ProcControl;
	pbMashPump : BOOL;
	PumpExp : BOOL;
	StartMash : BOOL;
	TimePre : DINT;
	MashACC : STRING[80];
	TmrRe : STRING[80];
	TmrRemain : STRING[80];
	CharNumPos : INT;
	MillNumPos : INT;
	NumStart : INT;
	TmrDT : TIMEStructure;
	RemainTime : DATE_AND_TIME;
	HrRe : STRING[4];
	MinRe : STRING[4];
	SecRe : STRING[4];
END_VAR
```

#### Main.st
```iecst
PROGRAM _INIT
	(* Insert code here *)

END_PROGRAM

PROGRAM _CYCLIC

		//Automatic and manual conditions
	mProc.Status.Automatic 	:= mProc.i.Start;
	mProc.Status.Manual		:= NOT mProc.i.Start;
	FromMashCyc.Start := mProc.i.Start;

	//Set the state machine
	IF  DiagCpuIsARsim() OR DiagCpuIsSimulated() THEN
		IF mProc.Status.Automatic THEN
			mProc.State := SimAuto;
		ELSIF mProc.Status.Manual THEN
			mProc.State := SimManual;
		END_IF
	END_IF

	//Turn off pump when switching auto and manual
	IF EDGENEG(mProc.i.Start) THEN
		pbMashPump 		:= FALSE;
		StartMash 		:= FALSE;
		MashTmr.IN		:= FALSE;
		mProc.i.Start 	:= FALSE;
	END_IF

	CASE mProc.State OF

		SimManual:
			//Figure out how to simulate the temperature
			mProc.currTemp := rawMashTemp / 1000;
			PumpExp := pbMashPump;

		SimAuto:
			//Figure out how to simulate the temperature
			mProc.currTemp := rawMashTemp / 1000;
			FromMashCyc.HLTTemp := mProc.SetTemp + 15;
			pbMashPump := PumpExp;

			//Stop pump if the mash temp gets too high
			IF mProc.currTemp < mProc.SetTemp THEN
				PumpExp	:= TRUE;
			ELSE
				PumpExp	:= FALSE;
			END_IF

			//Mash timer
			MashTmr.PT := DINT_TO_TIME(TimePre*60000);
			//Start Mash Timer
			MashTmr.IN := StartMash;

			//Calculate and display the remaining time
			TmrRe := TIME_TO_STRING(MashTmr.PT - MashTmr.ET);
			//Remove the T#
			TmrRemain := DELETE(TmrRe,2,1);
			// Find the first '_' in string
			TmrRemain := REPLACE(TmrRemain, ' ',1,FIND(TmrRemain,'_'));
			//Find the second '_' in string
			TmrRemain := REPLACE(TmrRemain, ' ',1,FIND(TmrRemain,'_'));
			//Remove everything after seconds
			TmrRemain := DELETE(TmrRemain,6,8);

			IF MashTmr.Q THEN
				StartMash := FALSE;
				mProc.i.Start := FALSE;
			END_IF

		Manual:

			mProc.currTemp := rawMashTemp / 1000;

	END_CASE

	MashPump := PumpExp;

	MashTmr();
END_PROGRAM

PROGRAM _EXIT
	(* Insert code here *)

END_PROGRAM
```

### Program Logical/TempControl/HLT (IEC)

#### Types.typ
```iecst
TYPE
	ControlState :
		(
		Manual,
		Automatic,
		SimManual,
		SimAuto
		);
	Controller : 	STRUCT
		ManPWM : MTBasicsPWM;
		State : ControlState;
		TempPram : MpTempControllerParType;
		TempCont : MpTempController;
	END_STRUCT;
END_TYPE
```

#### Variables.var
```iecst
VAR
	Proc : Controller;
END_VAR
```

#### Main.st
```iecst
PROGRAM _INIT

END_PROGRAM

PROGRAM _CYCLIC
	//Initilize Temp Controller FB
	Proc.TempCont.Parameters := ADR(Proc.TempPram);
	Proc.TempCont.MpLink := ADR(Cfg_HLTTemp);
	//Map Variables
	Proc.TempCont.Control := contHLT.Start;
	Proc.TempCont.ErrorReset := contHLT.ErrorReset;
	contHLT.Running := Proc.TempCont.ControlActive;

	//Set the state machine
	IF  DiagCpuIsARsim() OR DiagCpuIsSimulated() THEN
		IF sys.Stat.Automatic THEN
			Proc.State := SimAuto;
		ELSIF sys.Stat.Manual THEN
			Proc.State := SimManual;
		END_IF
	END_IF

	CASE Proc.State OF

		SimAuto:
			Proc.ManPWM.Enable := FALSE;
			Proc.TempCont.Enable := TRUE;
			Proc.TempCont.Simulate := TRUE;
			//Simulated Values
			Proc.TempCont.ActualTemperature := Proc.TempCont.Info.Simulation.ActualTemperature;
			Proc.TempCont.SetTemperature := contHLT.SetTemp;
			Proc.TempCont.Control := contHLT.Start;
			contHLT.Temperature := Proc.TempCont.Info.Simulation.ActualTemperature;
			contHLT.currPower := Proc.TempCont.Info.Simulation.HeatValue;

		SimManual:
			Proc.ManPWM.Enable := TRUE;
			Proc.TempCont.Enable := FALSE;
			//Proc.ManPWM Variables
			Proc.ManPWM.DutyCycle := contHLT.setPower;
			Proc.ManPWM.MinPulseWidth := 0.1;
			Proc.ManPWM.Period := 1.0;
			//contHLT.Temperature := contHLT.Temperature + 0.1;

		Automatic:
			Proc.ManPWM.Enable := TRUE;
			Proc.TempCont.Enable := FALSE;
			Proc.TempCont.ActualTemperature := rawHLTTemp * 1000;
			contHLT.currPower := Proc.TempCont.HeatValue;
			contHLT.Temperature := rawHLTTemp * 1000;
		Manual:
			Proc.ManPWM.Enable := FALSE;
			Proc.TempCont.Enable := TRUE;
			//Proc.ManPWM Variables
			Proc.ManPWM.DutyCycle := contHLT.setPower;
			Proc.ManPWM.MinPulseWidth := 0.1;
			Proc.ManPWM.Period := 1.0;
			contHLT.Temperature := rawHLTTemp * 1000;

	END_CASE

	//Call FB's
	Proc.TempCont();
	Proc.ManPWM();
END_PROGRAM

PROGRAM _EXIT
	(* Insert code here *)

END_PROGRAM
```

### Program Logical/TempControl/Kettle (IEC)

#### Variables.var
```iecst
VAR
	Mp_Parameters : MpTempControllerParType;
	Mp_Controller : MpTempController;
END_VAR
```

Listed in the project but not available here: Logical/Libraries/Functions/Types.typ, Logical/Libraries/Functions/Constants.var, Logical/Brewing/KettleControl/Types.typ, Logical/Distilling, Logical/Fermenting/Fermenting/Main.st, Logical/Fermenting/Fermenting/Types.typ, Logical/Fermenting/Fermenting/Variables.var
